// TIA Portal V20 export
DATA_BLOCK "CallEquipment_DB"   // DB80
{ DB_Accessible_From_OPC_UA := 'FALSE' }
// stored: AssignedProDiagFB Unit1.Em8.ProDiag, DBAccessibleFromOPCUA false, DBAccessibleFromWebserver false, InstanceOfName Unit1.Em8.CallEquipment, InstanceOfType FB, Namespace Unit1.Em8
"Unit1.Em8.CallEquipment"
   // VAR_INPUT
   //    ZoneOperationEnable { ExternalWritable := 'False'} : "LWONIK_typeSafetyZoneManualOperation";
   // END_VAR
   // VAR_IN_OUT
   //    unitStatus : "LAF_typeUnitStatus";
   //    emFeedback : "LUC_typeEmFeedback";
   //    unitAlarmDB : "LAF_typeAlarms";
   // END_VAR
   // VAR
   //    InstHipotThicknessSequence { ExternalWritable := 'False'} : "Unit1.Em8.Sequence_1_HipotThickness";
   //    InstHipotThicknessRnRSequence { S7_SetPoint := 'True'} : "Unit1.Em8.Sequence_10_GuageRnR";
   //    instHipotThicknessHomeJob1 { ExternalWritable := 'False'} : "LAF_SelectJob";
   //    instHipotThicknessLoadJob2 { ExternalWritable := 'False'} : "LAF_SelectJob";
   //    instHipotThicknessInspectionJob3 { ExternalWritable := 'False'} : "LAF_SelectJob";
   //    instHipotThicknessUnloadJob4 { ExternalWritable := 'False'} : "LAF_SelectJob";
   //    instGRnR_HipotThicknessLoad_Job2 { S7_SetPoint := 'True'} : "LAF_SelectJob";
   //    instGRnR_HipotThicknessInspection_Job3 { S7_SetPoint := 'True'} : "LAF_SelectJob";
   //    instGRnR_HipotThicknessUnload_Job4 { S7_SetPoint := 'True'} : "LAF_SelectJob";
   //    instCmHipotThicknessSafetyPin { ExternalWritable := 'False'} : "LBC_DigitalSignalCn";
   //    instCmHipotThicknessJRDetect { ExternalWritable := 'False'} : "LBC_DigitalSignalCn";
   //    instCmThicknessAxisZ { ExternalWritable := 'False'} : "LBC_Axis64Pos_TecPlcCn";
   //    instCmHipotThinknessStageLiftFrontUpDown { ExternalWritable := 'False'} : "LBC_TwoWayActuatorCn";
   //    instCmHipotThinknessStageLiftRearUpDown { ExternalWritable := 'False'} : "LBC_TwoWayActuatorCn";
   //    instCmHipotTabContactorBwdFwd { ExternalWritable := 'False'} : "LBC_TwoWayActuatorCn";
   //    instCmHipotTabContactorLeftOpenClose { ExternalWritable := 'False'} : "LBC_TwoWayActuatorCn";
   //    instCmHipotTabContactorRightOpenClose { ExternalWritable := 'False'} : "LBC_TwoWayActuatorCn";
   //    instCmHipotThinknessStageLiftAllUpDown { ExternalWritable := 'False'} : "LBC_TwoWayActuatorCn";
   //    instCmHipotControl { ExternalWritable := 'False'} : "LER_IRCheck_BT5525";
   //    instCmThicknessControl { ExternalWritable := 'False'} : "LER_Thickness";
   //    instCmHipotThicknessServoPress { ExternalWritable := 'False'} : "LER_ServoPress";
   //    instInterlockThicknessAxisZ { ExternalWritable := 'False'} : "LER_Axis64Pos_InterlockSummary";
   //    instLDrv701ControlThicknessAxisZ { ExternalWritable := 'False'} : "LDrvSafe_SinaTlg701Control";
   //    instLDrv701StatusThicknessAxisZ { ExternalWritable := 'False'} : "LDrvSafe_SinaTlg701Status";
   //    instHipotThicknessPressHistory { ExternalWritable := 'False'} : "LER_ServoPressHistory";
   //    instHipotHistory { ExternalWritable := 'False'} : "LER_hipotHistory";
   //    instThicknessHistory { ExternalWritable := 'False'} : "LER_thicknessHistory";
   //    instManageAlarms { ExternalWritable := 'False'} : "LAF_ManageAlarms";
   //    instEventsPFE { ExternalWritable := 'False'} : "Unit1.Em8.EventsPFE";
   //    statUnitStatus { ExternalWritable := 'False'} : "LAF_typeUnitStatus";
   //    statSlmStatus { ExternalWritable := 'False'} : Struct
   //       running : Bool;
   //       powerOff : Bool;
   //    END_STRUCT;
   //    statAllBrakeTest { ExternalWritable := 'False'} : "LER_typeBrakeTestUnitCommands";
   //    statPartData { ExternalWritable := 'False'} : "LER_typePartData";
   //    statDataDelete { ExternalWritable := 'False'} : "LER_typePartData";
   //    statHistoryDeleteData_press { ExternalWritable := 'False'} : "LER_typeServoPressHistory";
   //    statHistoryDeleteData_hipot { ExternalWritable := 'False'} : "LER_typeHipotHistory";
   //    statHistoryDeleteData_thickness { ExternalWritable := 'False'} : "LER_typeThicknessHistory";
   //    "statHistoryDeleteData_thicknessR&R" { ExternalWritable := 'False'} : "LER_typeThicknessHistory_R&R";
   //    statRoutingOk { ExternalWritable := 'False'} : Array[0..99] of Bool;
   //    statRoutingNok { ExternalWritable := 'False'} : Array[0..99] of Bool;
   //    statTonTime { ExternalWritable := 'False'} : Array[0..999] of TON_TIME;
   //    statTofTime { ExternalWritable := 'False'} : Array[0..9] of TOF_TIME;
   //    statPulse { ExternalWritable := 'False'} : Array[0..999] of Bool;
   //    statGaugeRnR { ExternalWritable := 'False'} : Struct
   //       currentCount : Int;
   //       processCount : Int := 50;
   //       Ongoing : Bool;
   //       Complete : Bool;
   //    END_STRUCT;
   //    statEnableManualCmds { ExternalWritable := 'False'} : Bool;
   //    statNomalMode { ExternalWritable := 'False'} : Bool;
   //    "*** Interlock Axis ***" : Bool;
   //    ThicknessAxisZ_Jog { S7_SetPoint := 'True'} : Array[0..2] of "LER_Axis_Jog";
   //    ThicknessAxisZ_interlock { S7_SetPoint := 'True'} : Array[0..10] of "LER_Axis_Absolute";
   //    ThicknessAxisZ_IntPos : Array[0..9] of Struct
   //       "Int" : Array[1..10] of Bool;
   //    END_STRUCT;
   //    ThicknessAxisZ_IntHome : Array[0..9] of Bool;
   //    ThicknessAxisZ_PosAbsolute : Array[0..10] of Bool;
   //    ThicknessAxisZ_Home { S7_SetPoint := 'True'} : "LER_Axis_Homing";
   //    "*** Interlock TwoWay ***" { S7_SetPoint := 'True'} : "LER_Axis_Homing";
   //    instCmHipotThinknessStageLiftFrontUpDownInterlock { S7_SetPoint := 'True'} : Array[0..2] of "LER_Actuator";
   //    instCmHipotThinknessStageLiftRearUpDownInterlock { S7_SetPoint := 'True'} : Array[0..2] of "LER_Actuator";
   //    instCmHipotTabContactorBwdFwdInterlock { S7_SetPoint := 'True'} : Array[0..2] of "LER_Actuator";
   //    instCmHipotTabContactorLeftOpenCloseInterlock { S7_SetPoint := 'True'} : Array[0..2] of "LER_Actuator";
   //    instCmHipotTabContactorRightOpenCloseInterlock { S7_SetPoint := 'True'} : Array[0..2] of "LER_Actuator";
   //    instCmHipotThinknessStageLiftAllUpDownInterlock { S7_SetPoint := 'True'} : Array[0..2] of "LER_Actuator";
   //    HipotThinknessStageLiftFrontUpDown_Inpos : Array[0..2] of Struct
   //       "Int" : Array[1..10] of Bool;
   //    END_STRUCT;
   //    HipotThinknessStageLiftRearUpDown_Inpos : Array[0..2] of Struct
   //       "Int" : Array[1..10] of Bool;
   //    END_STRUCT;
   //    HipotTabContactorBwdFwd_Inpos : Array[0..2] of Struct
   //       "Int" : Array[1..10] of Bool;
   //    END_STRUCT;
   //    HipotTabContactorLeftOpenClose_Inpos : Array[0..2] of Struct
   //       "Int" : Array[1..10] of Bool;
   //    END_STRUCT;
   //    HipotTabContactorRightOpenClose_Inpos : Array[0..2] of Struct
   //       "Int" : Array[1..10] of Bool;
   //    END_STRUCT;
   //    HipotThinknessStageLiftAllUpDown_Inpos : Array[0..2] of Struct
   //       "Int" : Array[1..10] of Bool;
   //    END_STRUCT;
   //    citi_Ptrig : Array[0..20] of Bool;
   //    citiTon : Array[0..20] of TON_TIME;
   //    citi : Time;
   //    citiTest : Array[0..20] of Bool;
   //    instPFERecipe { S7_SetPoint := 'True'} : "Unit1.Em8.EventsPFE_Recipe";
   // END_VAR
BEGIN
END_DATA_BLOCK
